FUNCTION_BLOCK System_IpcInfo
VAR_INPUT
END_VAR
VAR_OUTPUT
END_VAR
VAR
END_VAR

END_FUNCTION_BLOCK

(* stored: Version 1.1.0.1, ProductVersion 3.1.4024.12
   POU System_IpcInfo: Id {6baa2aa1-d5d7-4b2b-87dd-5d6201c5627a}, SpecialFunc None *)
